(* PLC project model, Beckhoff Automation Beckhoff MLlib 3.1.251201.0 *)
(* stored: creationDateTime 2026-07-10T12:15:14.2510637, modificationDateTime 2026-07-10T12:15:14.2510637 *)

TYPE ST_modelInput :
STRUCT

	{attribute 'hide'} _header_DO_NOT_CHANGE : ARRAY[0..63] OF SINT := [-1,-112,120,86,52,18,-1,-1,1,-1,0,0,-1,-1,-112,-112,61,-49,110,-13,101,63,-28,35,-75,-48,62,84,75,113,93,86,13,-100,61,-11,-76,-124,91,74,-32,110,127,-106,67,10,-85,-84,84,0,0,0,0,0,0,0,0,0,0,0,0,0,0,0];
	in_input_tensor : ARRAY[0..0,0..4] OF REAL;

END_STRUCT
END_TYPE

TYPE ST_modelOutput :
STRUCT

	{attribute 'hide'} _header_DO_NOT_CHANGE : ARRAY[0..63] OF SINT := [-1,-112,120,86,52,18,-1,-1,1,-1,0,0,-1,-1,-112,-112,-35,24,-50,75,-65,96,-121,123,127,87,61,127,-39,-108,16,-70,120,-89,-28,78,-43,26,-32,-7,81,19,29,-89,-55,3,43,2,68,0,0,0,0,0,0,0,0,0,0,0,0,0,0,0];
	out_prediction_tensor : ARRAY[0..0,0..0] OF REAL;

END_STRUCT
END_TYPE
